// TIA Portal V16 export
// export: Created 2022-07-21T09:35:28.7234867Z, ExportSetting WithDefaults, DisplayName Totally Integrated Automation Portal, DisplayVersion V16 Update 4, DisplayName TIA Portal Version Control Interface, DisplayVersion V16 Update 2, DisplayName TIA Portal Openness, DisplayVersion V16 Update 4, DisplayName SINAMICS Startdrive Advanced, DisplayVersion V16 Update 5, DisplayName SINAMICS Startdrive G130, G150, S120, S150, SINAMICS MV, S210, DisplayVersion V16 Update 5, DisplayName SINAMICS Startdrive G110M, G120, G120C, G120D, G120P, G115D, DisplayVersion V16 Update 5, DisplayName STEP 7 Professional, DisplayVersion V16 Update 4, DisplayName STEP 7 Safety, DisplayVersion V16, DisplayName WinCC Advanced, DisplayVersion V16 Update 4
FUNCTION "fcPowerUnit" : Void   // FC31, LAD
{ S7_Optimized_Access := 'TRUE' }
VERSION : 0.1
// stored: AutoNumber true, IsIECCheckEnabled false, SetENOAutomatically false, UDAEnableTagReadback false
   VAR_INPUT
      inEnable : Bool;
      inDisable : Bool;
      inReset : Bool;
   END_VAR
   VAR_OUTPUT
      ouEnable : Bool;
      ouDisable : Bool;
      ouReset : Bool;
   END_VAR
BEGIN

REGION Network 1: Załączenie stycznika mocy
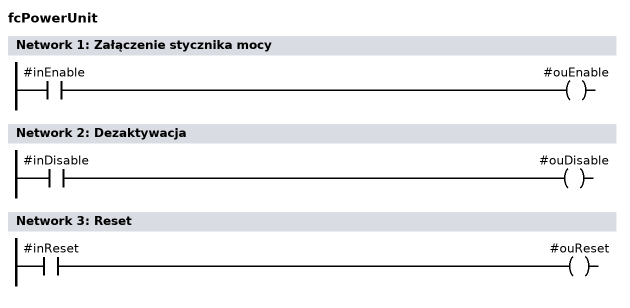
   RUNG wire#powerrail
      Contact( #inEnable )
      Coil( #ouEnable )
   END_RUNG
   // the same network as SCL:
   #ouEnable := #inEnable;
END_REGION

REGION Network 2: Dezaktywacja
   RUNG wire#powerrail
      Contact( #inDisable )
      Coil( #ouDisable )
   END_RUNG
   // the same network as SCL:
   #ouDisable := #inDisable;
END_REGION

REGION Network 3: Reset
   RUNG wire#powerrail
      Contact( #inReset )
      Coil( #ouReset )
   END_RUNG
   // the same network as SCL:
   #ouReset := #inReset;
END_REGION
END_FUNCTION
